(* Logix 5000 project; controller BreakGroup_US vendor 1 type 14 code 211 rev 32.16; software revision 32.05; part 5 of 8 *)
(* tags used below, declared in another part *)
   Emg_Stop : BOOL;
   Gantry_2_Tilter_LH_Start : BOOL;
   HMI_MAN_LH_OIL_STOP : BOOL;
   HMI_MAN_RH_OIL_STOP : BOOL;
   HMI_MAN_STN_100_STOP : BOOL;
   HMI_MAN_STN_110_STOP : BOOL;
   HMI_Oil_Tank_LH_PB : SINT;
   HMI_Oil_Tank_RH_PB : SINT;
   MAN_LH_OIL_TIME : TIMER;
   MAN_RH_OIL_TIME : TIMER;
   MAN_STN_100_HOME : TIMER;
   MAN_STN_110_HOME : TIMER;
   MCP_GY_01_Gripper : MCP_Servo_01;
   MCP_GY_01_Horizontal : MCP_Servo_02;
   MCP_GY_01_Vertical : MCP_Servo_02;
   RCP_LH_Oil_Tank_Lift : RCP_Servo_02;
   RCP_LH_Oil_Tank_Lift_Start : BOOL;
   RCP_RH_Oil_Tank_Lift : RCP_Servo_02;
   RCP_RH_Oil_Tank_Lift_Start : BOOL;
   RCP_ST_100_Turntable_Motor : RCP_Servo_02;
   RCP_ST_110_Turntable_Motor : RCP_Servo_02;
   ST10_Pre_Condition_OK : BOOL;
   ST10_Trolley1Lock_Cyl_01_Extended : ALIAS FOR MCP_PT01:1:I.0;
   ST10_Trolley1LockCyl_01_Retracted : ALIAS FOR MCP_PT01:1:I.1;
   ST10_Trolley_Present_Sensor : ALIAS FOR MCP_PT01:1:I.2;
   ST_100_Start : BOOL;
   ST_10_SEQ : DINT;
   ST_10_T1 : TIMER;
   ST_10_Trolley_FRWD : BOOL;
   ST_110_Start : BOOL;
   STN_100_Connection_Fault : BOOL;
   STN_100_Conveyor : INDEX_Block;
   STN_100_HMI_PB : SINT[2];
   STN_110_Connection_fault : BOOL;
   STN_110_Conveyor : INDEX_Block;
   STN_110_HMI_PB : SINT[2];

PROGRAM Oil_Tank_Lift   (* main routine Main *)

ROUTINE Main   (* ladder *)
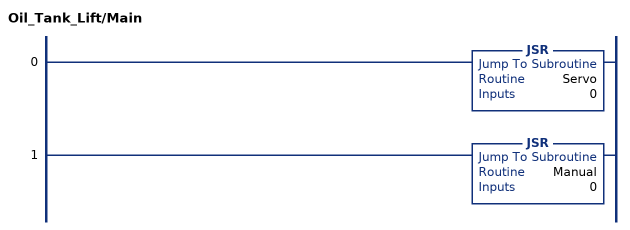
   0: JSR(Servo,0);
   1: JSR(Manual,0);
END_ROUTINE

ROUTINE Manual   (* ladder *)
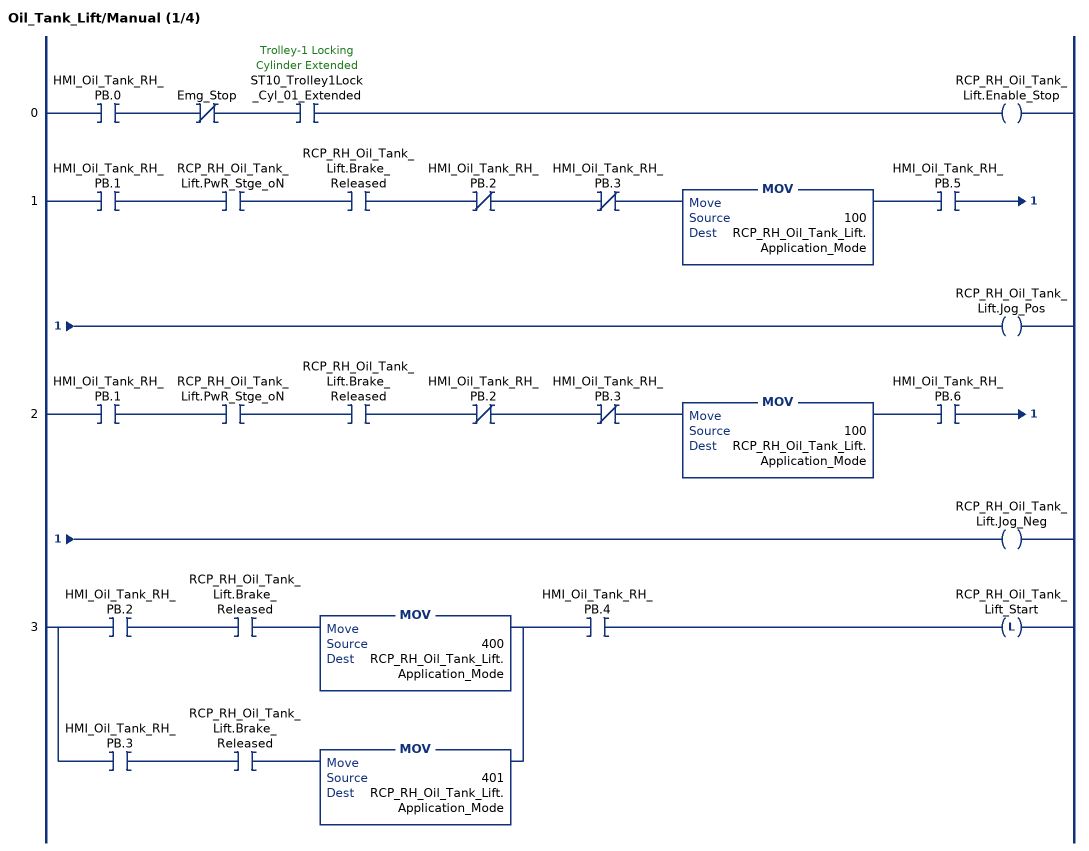
   0: XIC(HMI_Oil_Tank_RH_PB.0)XIO(Emg_Stop)XIC(ST10_Trolley1Lock_Cyl_01_Extended)OTE(RCP_RH_Oil_Tank_Lift.Enable_Stop);
   1: XIC(HMI_Oil_Tank_RH_PB.1)XIC(RCP_RH_Oil_Tank_Lift.PwR_Stge_oN)XIC(RCP_RH_Oil_Tank_Lift.Brake_Released)XIO(HMI_Oil_Tank_RH_PB.2)XIO(HMI_Oil_Tank_RH_PB.3)MOV(100,RCP_RH_Oil_Tank_Lift.Application_Mode)XIC(HMI_Oil_Tank_RH_PB.5)OTE(RCP_RH_Oil_Tank_Lift.Jog_Pos);
   2: XIC(HMI_Oil_Tank_RH_PB.1)XIC(RCP_RH_Oil_Tank_Lift.PwR_Stge_oN)XIC(RCP_RH_Oil_Tank_Lift.Brake_Released)XIO(HMI_Oil_Tank_RH_PB.2)XIO(HMI_Oil_Tank_RH_PB.3)MOV(100,RCP_RH_Oil_Tank_Lift.Application_Mode)XIC(HMI_Oil_Tank_RH_PB.6)OTE(RCP_RH_Oil_Tank_Lift.Jog_Neg);
   3: [XIC(HMI_Oil_Tank_RH_PB.2) XIC(RCP_RH_Oil_Tank_Lift.Brake_Released) MOV(400,RCP_RH_Oil_Tank_Lift.Application_Mode) ,XIC(HMI_Oil_Tank_RH_PB.3) XIC(RCP_RH_Oil_Tank_Lift.Brake_Released) MOV(401,RCP_RH_Oil_Tank_Lift.Application_Mode) ]XIC(HMI_Oil_Tank_RH_PB.4)OTL(RCP_RH_Oil_Tank_Lift_Start);
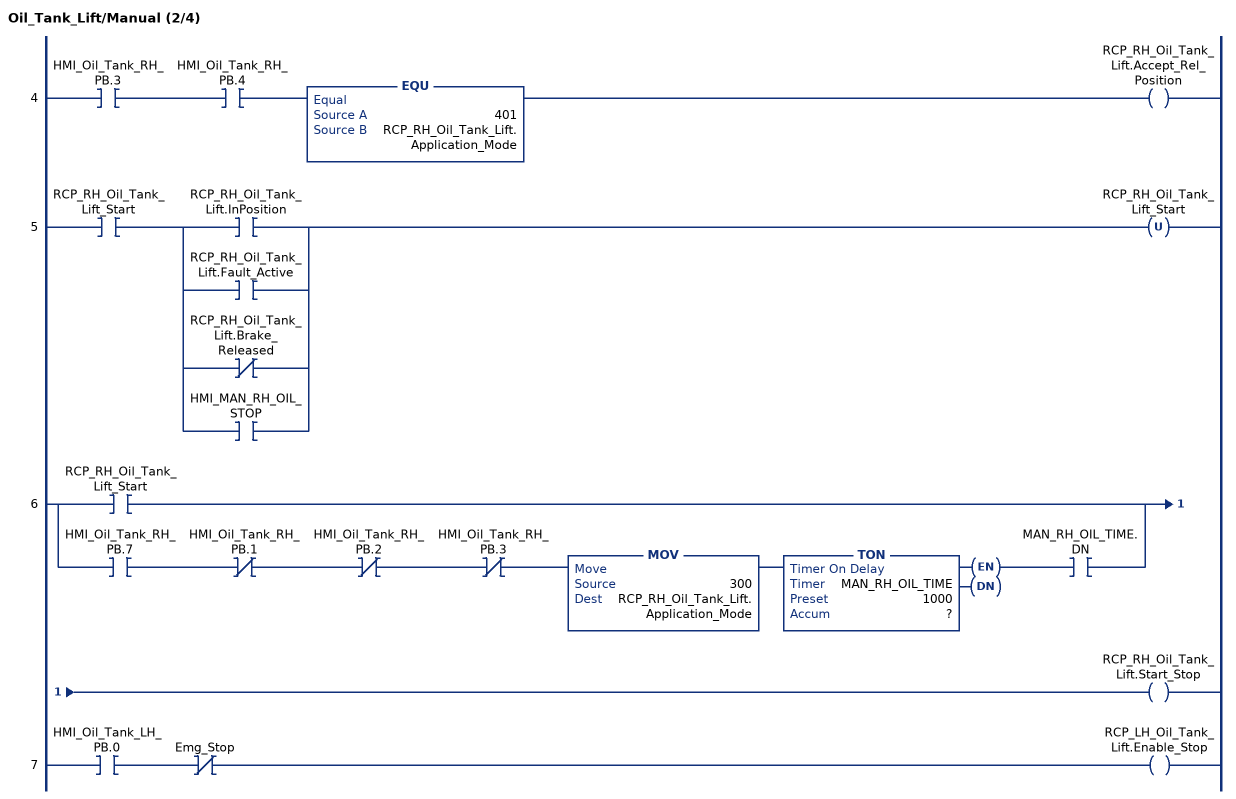
   4: XIC(HMI_Oil_Tank_RH_PB.3)XIC(HMI_Oil_Tank_RH_PB.4)EQU(401,RCP_RH_Oil_Tank_Lift.Application_Mode)OTE(RCP_RH_Oil_Tank_Lift.Accept_Rel_Position);
   5: XIC(RCP_RH_Oil_Tank_Lift_Start)[XIC(RCP_RH_Oil_Tank_Lift.InPosition) ,[XIC(RCP_RH_Oil_Tank_Lift.Fault_Active) ,[XIO(RCP_RH_Oil_Tank_Lift.Brake_Released) ,XIC(HMI_MAN_RH_OIL_STOP) ] ] ]OTU(RCP_RH_Oil_Tank_Lift_Start);
   6: [XIC(RCP_RH_Oil_Tank_Lift_Start) ,XIC(HMI_Oil_Tank_RH_PB.7) XIO(HMI_Oil_Tank_RH_PB.1) XIO(HMI_Oil_Tank_RH_PB.2) XIO(HMI_Oil_Tank_RH_PB.3) MOV(300,RCP_RH_Oil_Tank_Lift.Application_Mode) TON(MAN_RH_OIL_TIME,?,?) XIC(MAN_RH_OIL_TIME.DN) ]OTE(RCP_RH_Oil_Tank_Lift.Start_Stop);
   7: XIC(HMI_Oil_Tank_LH_PB.0)XIO(Emg_Stop)OTE(RCP_LH_Oil_Tank_Lift.Enable_Stop);
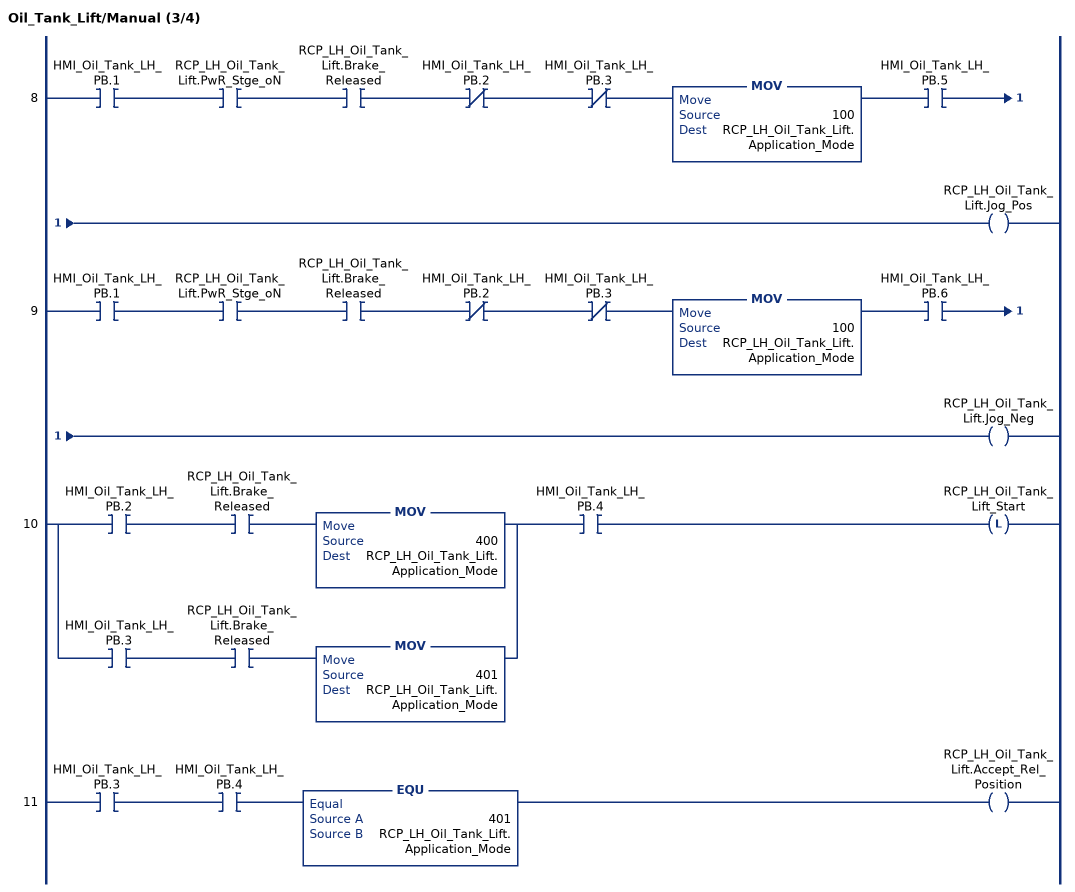
   8: XIC(HMI_Oil_Tank_LH_PB.1)XIC(RCP_LH_Oil_Tank_Lift.PwR_Stge_oN)XIC(RCP_LH_Oil_Tank_Lift.Brake_Released)XIO(HMI_Oil_Tank_LH_PB.2)XIO(HMI_Oil_Tank_LH_PB.3)MOV(100,RCP_LH_Oil_Tank_Lift.Application_Mode)XIC(HMI_Oil_Tank_LH_PB.5)OTE(RCP_LH_Oil_Tank_Lift.Jog_Pos);
   9: XIC(HMI_Oil_Tank_LH_PB.1)XIC(RCP_LH_Oil_Tank_Lift.PwR_Stge_oN)XIC(RCP_LH_Oil_Tank_Lift.Brake_Released)XIO(HMI_Oil_Tank_LH_PB.2)XIO(HMI_Oil_Tank_LH_PB.3)MOV(100,RCP_LH_Oil_Tank_Lift.Application_Mode)XIC(HMI_Oil_Tank_LH_PB.6)OTE(RCP_LH_Oil_Tank_Lift.Jog_Neg);
   10: [XIC(HMI_Oil_Tank_LH_PB.2) XIC(RCP_LH_Oil_Tank_Lift.Brake_Released) MOV(400,RCP_LH_Oil_Tank_Lift.Application_Mode) ,XIC(HMI_Oil_Tank_LH_PB.3) XIC(RCP_LH_Oil_Tank_Lift.Brake_Released) MOV(401,RCP_LH_Oil_Tank_Lift.Application_Mode) ]XIC(HMI_Oil_Tank_LH_PB.4)OTL(RCP_LH_Oil_Tank_Lift_Start);
   11: XIC(HMI_Oil_Tank_LH_PB.3)XIC(HMI_Oil_Tank_LH_PB.4)EQU(401,RCP_LH_Oil_Tank_Lift.Application_Mode)OTE(RCP_LH_Oil_Tank_Lift.Accept_Rel_Position);
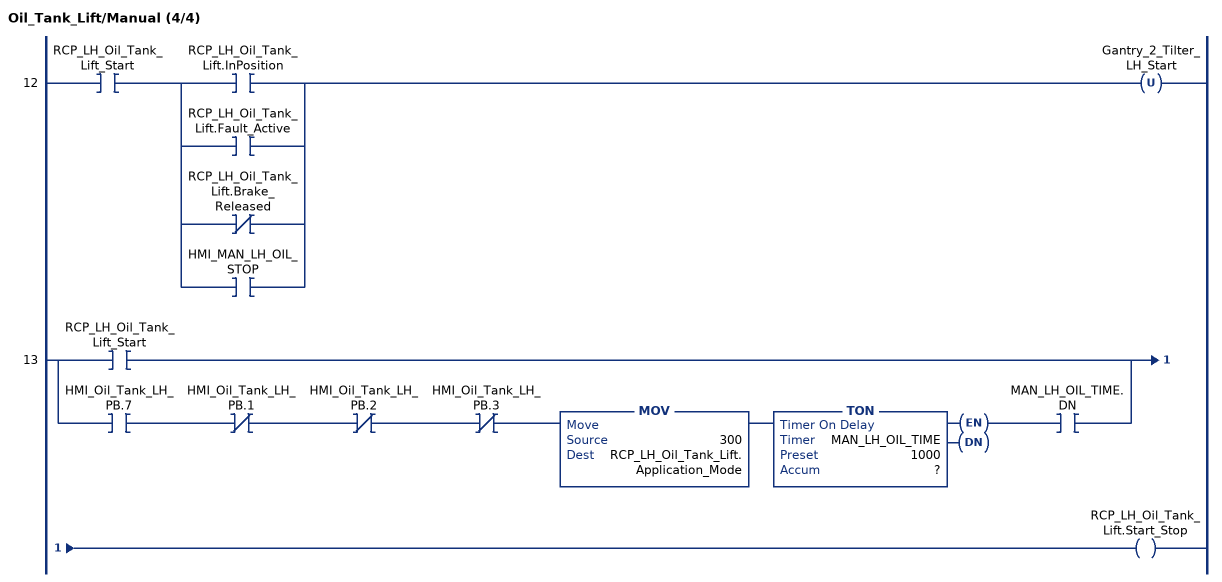
   12: XIC(RCP_LH_Oil_Tank_Lift_Start)[XIC(RCP_LH_Oil_Tank_Lift.InPosition) ,[XIC(RCP_LH_Oil_Tank_Lift.Fault_Active) ,[XIO(RCP_LH_Oil_Tank_Lift.Brake_Released) ,XIC(HMI_MAN_LH_OIL_STOP) ] ] ]OTU(Gantry_2_Tilter_LH_Start);
   13: [XIC(RCP_LH_Oil_Tank_Lift_Start) ,XIC(HMI_Oil_Tank_LH_PB.7) XIO(HMI_Oil_Tank_LH_PB.1) XIO(HMI_Oil_Tank_LH_PB.2) XIO(HMI_Oil_Tank_LH_PB.3) MOV(300,RCP_LH_Oil_Tank_Lift.Application_Mode) TON(MAN_LH_OIL_TIME,?,?) XIC(MAN_LH_OIL_TIME.DN) ]OTE(RCP_LH_Oil_Tank_Lift.Start_Stop);
END_ROUTINE

ROUTINE Servo   (* ladder *)
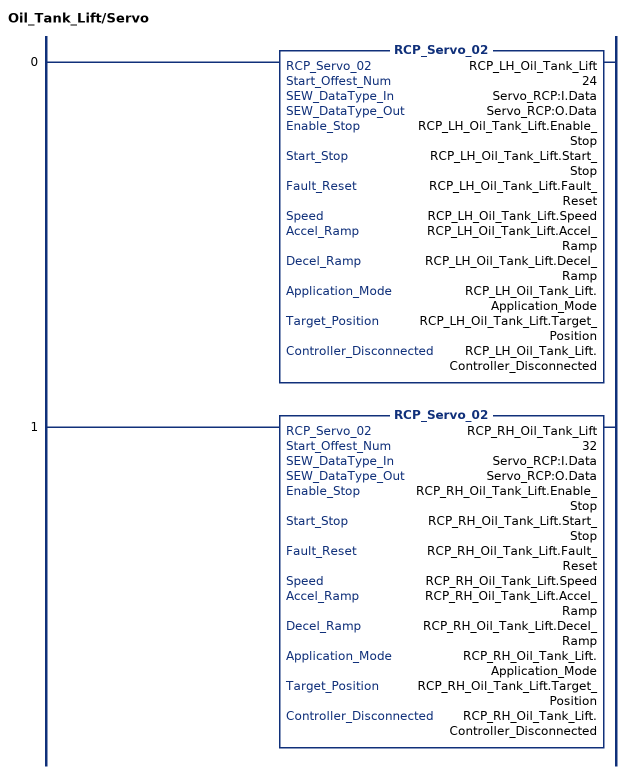
   0: RCP_Servo_02(RCP_LH_Oil_Tank_Lift,24,Servo_RCP:I.Data,Servo_RCP:O.Data,RCP_LH_Oil_Tank_Lift.Enable_Stop,RCP_LH_Oil_Tank_Lift.Start_Stop,RCP_LH_Oil_Tank_Lift.Fault_Reset,RCP_LH_Oil_Tank_Lift.Speed,RCP_LH_Oil_Tank_Lift.Accel_Ramp,RCP_LH_Oil_Tank_Lift.Decel_Ramp,RCP_LH_Oil_Tank_Lift.Application_Mode,RCP_LH_Oil_Tank_Lift.Target_Position,RCP_LH_Oil_Tank_Lift.Controller_Disconnected);
   1: RCP_Servo_02(RCP_RH_Oil_Tank_Lift,32,Servo_RCP:I.Data,Servo_RCP:O.Data,RCP_RH_Oil_Tank_Lift.Enable_Stop,RCP_RH_Oil_Tank_Lift.Start_Stop,RCP_RH_Oil_Tank_Lift.Fault_Reset,RCP_RH_Oil_Tank_Lift.Speed,RCP_RH_Oil_Tank_Lift.Accel_Ramp,RCP_RH_Oil_Tank_Lift.Decel_Ramp,RCP_RH_Oil_Tank_Lift.Application_Mode,RCP_RH_Oil_Tank_Lift.Target_Position,RCP_RH_Oil_Tank_Lift.Controller_Disconnected);
END_ROUTINE
END_PROGRAM

PROGRAM SafetyProgram   (* main routine MainRoutine, safety *)

ROUTINE MainRoutine   (* ladder *)
END_ROUTINE
END_PROGRAM

PROGRAM Station_10   (* main routine Main *)

ROUTINE Main   (* ladder *)
END_ROUTINE

ROUTINE Sequence   (* ladder *)
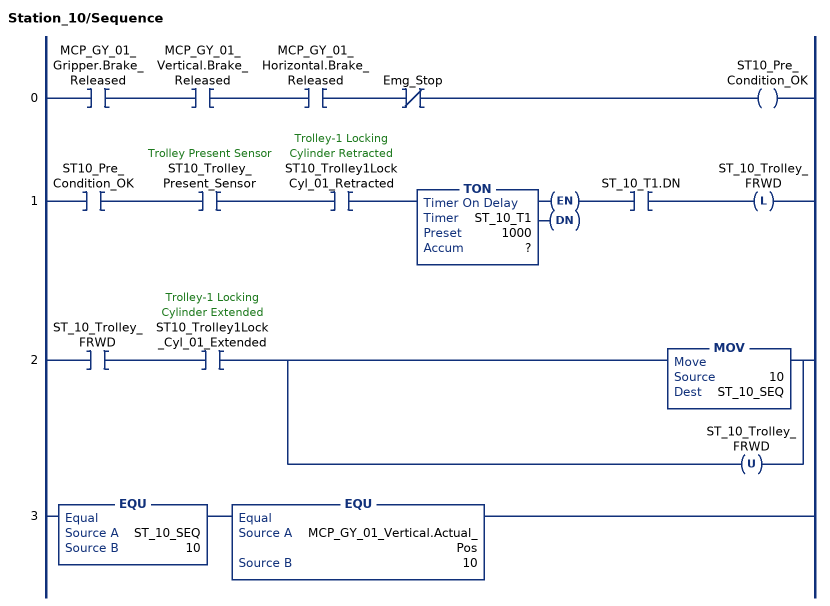
   0: XIC(MCP_GY_01_Gripper.Brake_Released)XIC(MCP_GY_01_Vertical.Brake_Released)XIC(MCP_GY_01_Horizontal.Brake_Released)XIO(Emg_Stop)OTE(ST10_Pre_Condition_OK);
   1: XIC(ST10_Pre_Condition_OK)XIC(ST10_Trolley_Present_Sensor)XIC(ST10_Trolley1LockCyl_01_Retracted)TON(ST_10_T1,?,?)XIC(ST_10_T1.DN)OTL(ST_10_Trolley_FRWD);
   2: XIC(ST_10_Trolley_FRWD)XIC(ST10_Trolley1Lock_Cyl_01_Extended)[MOV(10,ST_10_SEQ) ,OTU(ST_10_Trolley_FRWD) ];
   3: EQU(ST_10_SEQ,10)EQU(MCP_GY_01_Vertical.Actual_Pos,10);
END_ROUTINE
END_PROGRAM

PROGRAM Station_100   (* main routine Main *)

ROUTINE Main   (* ladder *)
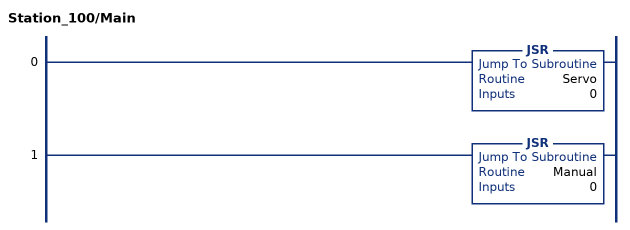
   0: JSR(Servo,0);
   1: JSR(Manual,0);
END_ROUTINE

ROUTINE Manual   (* ladder *)
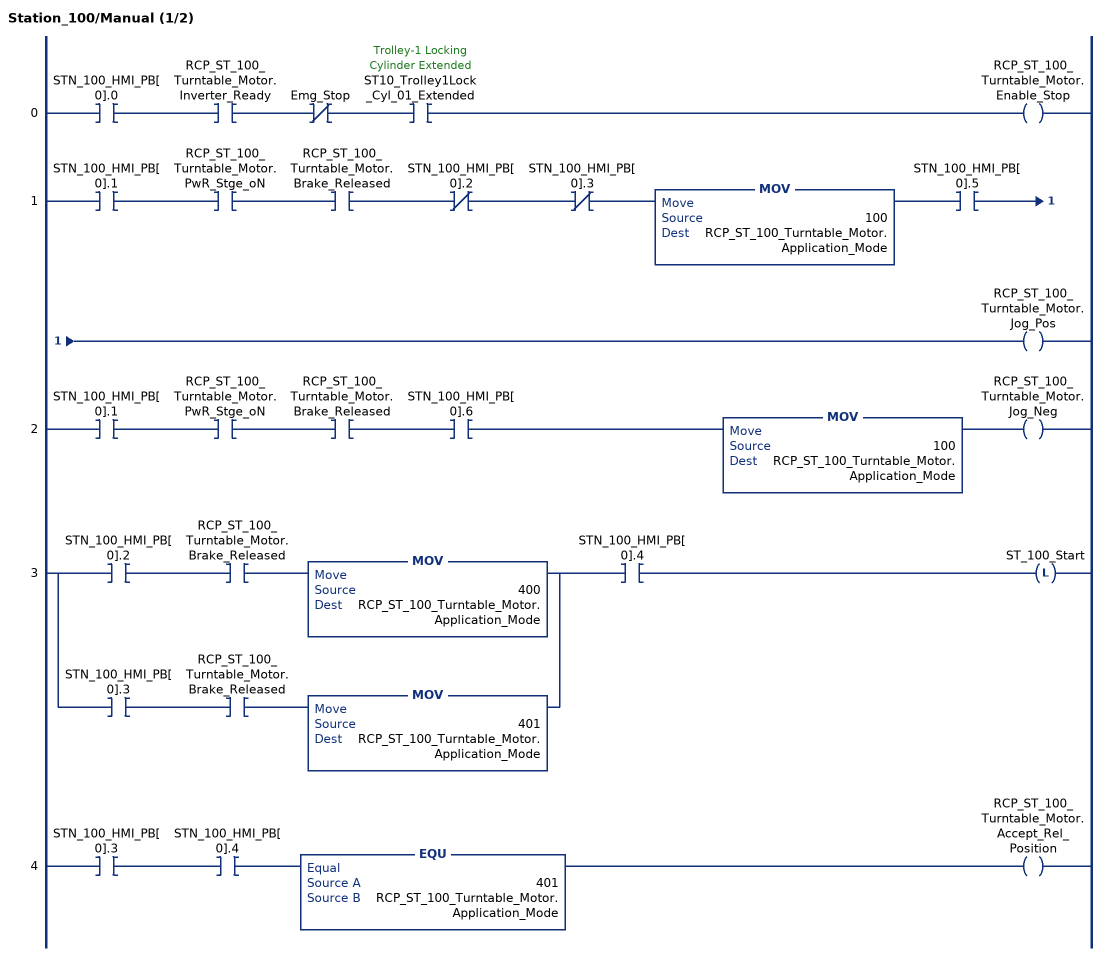
   0: XIC(STN_100_HMI_PB[0].0)XIC(RCP_ST_100_Turntable_Motor.Inverter_Ready)XIO(Emg_Stop)XIC(ST10_Trolley1Lock_Cyl_01_Extended)OTE(RCP_ST_100_Turntable_Motor.Enable_Stop);
   1: XIC(STN_100_HMI_PB[0].1)XIC(RCP_ST_100_Turntable_Motor.PwR_Stge_oN)XIC(RCP_ST_100_Turntable_Motor.Brake_Released)XIO(STN_100_HMI_PB[0].2)XIO(STN_100_HMI_PB[0].3)MOV(100,RCP_ST_100_Turntable_Motor.Application_Mode)XIC(STN_100_HMI_PB[0].5)OTE(RCP_ST_100_Turntable_Motor.Jog_Pos);
   2: XIC(STN_100_HMI_PB[0].1)XIC(RCP_ST_100_Turntable_Motor.PwR_Stge_oN)XIC(RCP_ST_100_Turntable_Motor.Brake_Released)XIC(STN_100_HMI_PB[0].6)MOV(100,RCP_ST_100_Turntable_Motor.Application_Mode)OTE(RCP_ST_100_Turntable_Motor.Jog_Neg);
   3: [XIC(STN_100_HMI_PB[0].2) XIC(RCP_ST_100_Turntable_Motor.Brake_Released) MOV(400,RCP_ST_100_Turntable_Motor.Application_Mode) ,XIC(STN_100_HMI_PB[0].3) XIC(RCP_ST_100_Turntable_Motor.Brake_Released) MOV(401,RCP_ST_100_Turntable_Motor.Application_Mode) ]XIC(STN_100_HMI_PB[0].4)OTL(ST_100_Start);
   4: XIC(STN_100_HMI_PB[0].3)XIC(STN_100_HMI_PB[0].4)EQU(401,RCP_ST_100_Turntable_Motor.Application_Mode)OTE(RCP_ST_100_Turntable_Motor.Accept_Rel_Position);
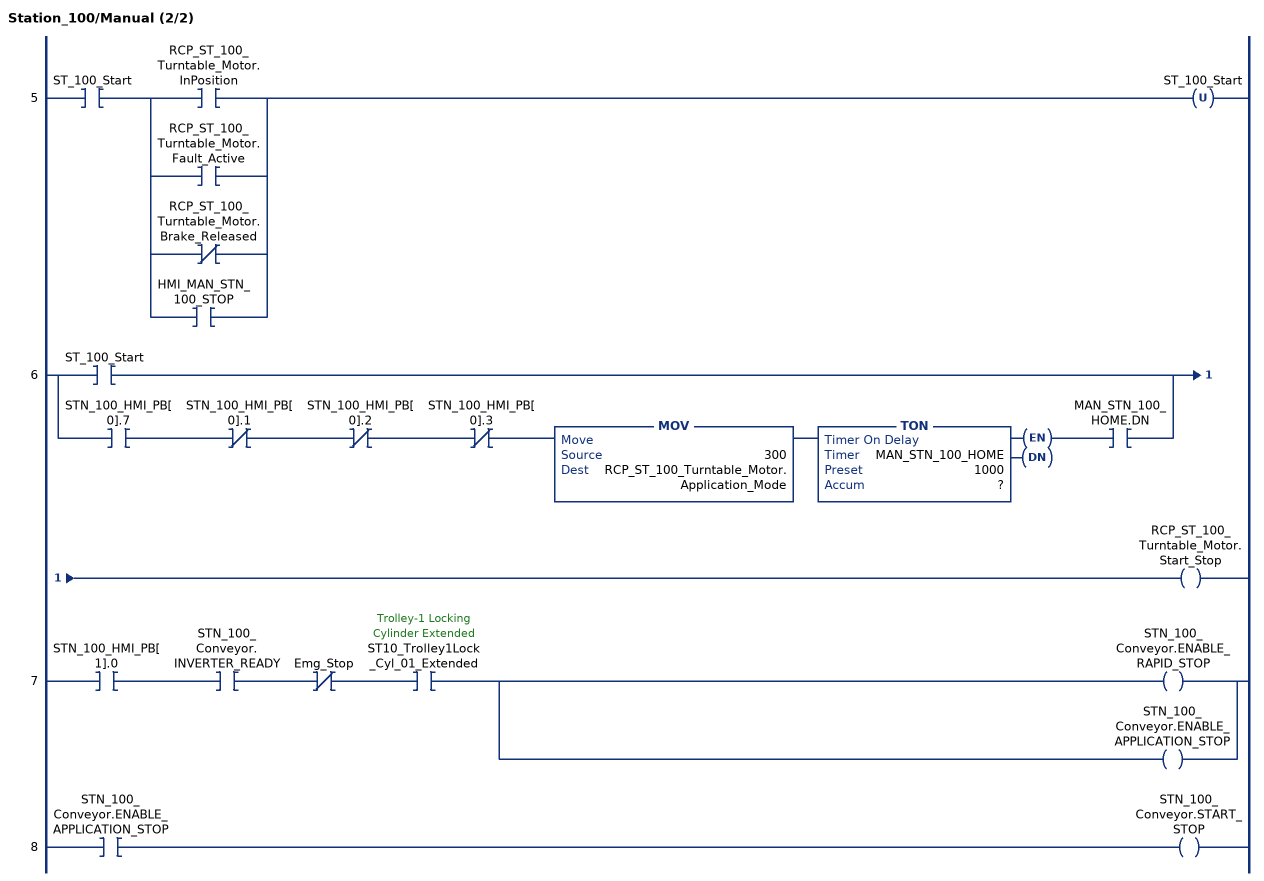
   5: XIC(ST_100_Start)[XIC(RCP_ST_100_Turntable_Motor.InPosition) ,[XIC(RCP_ST_100_Turntable_Motor.Fault_Active) ,[XIO(RCP_ST_100_Turntable_Motor.Brake_Released) ,XIC(HMI_MAN_STN_100_STOP) ] ] ]OTU(ST_100_Start);
   6: [XIC(ST_100_Start) ,XIC(STN_100_HMI_PB[0].7) XIO(STN_100_HMI_PB[0].1) XIO(STN_100_HMI_PB[0].2) XIO(STN_100_HMI_PB[0].3) MOV(300,RCP_ST_100_Turntable_Motor.Application_Mode) TON(MAN_STN_100_HOME,?,?) XIC(MAN_STN_100_HOME.DN) ]OTE(RCP_ST_100_Turntable_Motor.Start_Stop);
   7: XIC(STN_100_HMI_PB[1].0)XIC(STN_100_Conveyor.INVERTER_READY)XIO(Emg_Stop)XIC(ST10_Trolley1Lock_Cyl_01_Extended)[OTE(STN_100_Conveyor.ENABLE_RAPID_STOP) ,OTE(STN_100_Conveyor.ENABLE_APPLICATION_STOP) ];
   8: XIC(STN_100_Conveyor.ENABLE_APPLICATION_STOP)OTE(STN_100_Conveyor.START_STOP);
END_ROUTINE

ROUTINE Servo   (* ladder *)
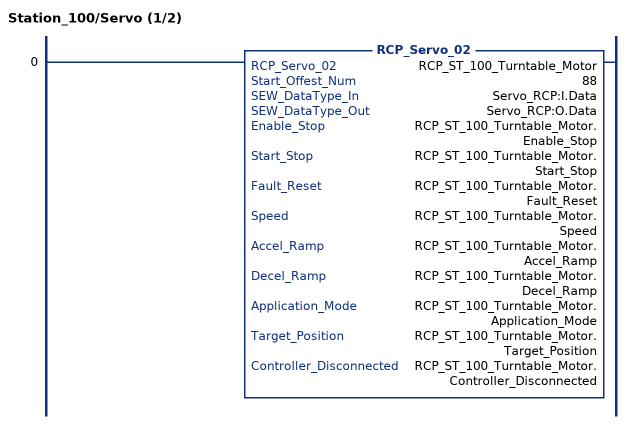
   0: RCP_Servo_02(RCP_ST_100_Turntable_Motor,88,Servo_RCP:I.Data,Servo_RCP:O.Data,RCP_ST_100_Turntable_Motor.Enable_Stop,RCP_ST_100_Turntable_Motor.Start_Stop,RCP_ST_100_Turntable_Motor.Fault_Reset,RCP_ST_100_Turntable_Motor.Speed,RCP_ST_100_Turntable_Motor.Accel_Ramp,RCP_ST_100_Turntable_Motor.Decel_Ramp,RCP_ST_100_Turntable_Motor.Application_Mode,RCP_ST_100_Turntable_Motor.Target_Position,RCP_ST_100_Turntable_Motor.Controller_Disconnected);
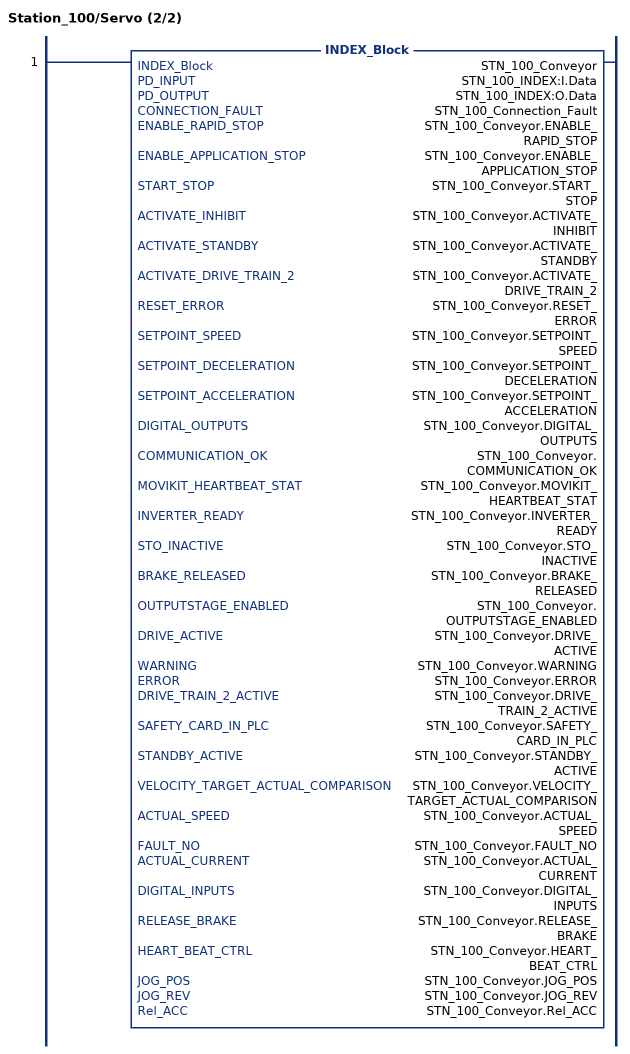
   1: INDEX_Block(STN_100_Conveyor,STN_100_INDEX:I.Data,STN_100_INDEX:O.Data,STN_100_Connection_Fault,STN_100_Conveyor.ENABLE_RAPID_STOP,STN_100_Conveyor.ENABLE_APPLICATION_STOP,STN_100_Conveyor.START_STOP,STN_100_Conveyor.ACTIVATE_INHIBIT,STN_100_Conveyor.ACTIVATE_STANDBY,STN_100_Conveyor.ACTIVATE_DRIVE_TRAIN_2,STN_100_Conveyor.RESET_ERROR,STN_100_Conveyor.SETPOINT_SPEED,STN_100_Conveyor.SETPOINT_DECELERATION,STN_100_Conveyor.SETPOINT_ACCELERATION,STN_100_Conveyor.DIGITAL_OUTPUTS,STN_100_Conveyor.COMMUNICATION_OK,STN_100_Conveyor.MOVIKIT_HEARTBEAT_STAT,STN_100_Conveyor.INVERTER_READY,STN_100_Conveyor.STO_INACTIVE,STN_100_Conveyor.BRAKE_RELEASED,STN_100_Conveyor.OUTPUTSTAGE_ENABLED,STN_100_Conveyor.DRIVE_ACTIVE,STN_100_Conveyor.WARNING,STN_100_Conveyor.ERROR,STN_100_Conveyor.DRIVE_TRAIN_2_ACTIVE,STN_100_Conveyor.SAFETY_CARD_IN_PLC,STN_100_Conveyor.STANDBY_ACTIVE,STN_100_Conveyor.VELOCITY_TARGET_ACTUAL_COMPARISON,STN_100_Conveyor.ACTUAL_SPEED,STN_100_Conveyor.FAULT_NO,STN_100_Conveyor.ACTUAL_CURRENT,STN_100_Conveyor.DIGITAL_INPUTS,STN_100_Conveyor.RELEASE_BRAKE,STN_100_Conveyor.HEART_BEAT_CTRL,STN_100_Conveyor.JOG_POS,STN_100_Conveyor.JOG_REV,STN_100_Conveyor.Rel_ACC);
END_ROUTINE
END_PROGRAM

PROGRAM Station_110   (* main routine Main *)

ROUTINE Main   (* ladder *)
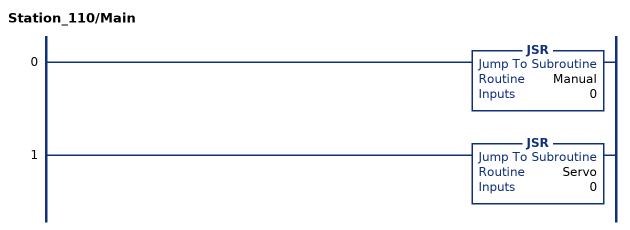
   0: JSR(Manual,0);
   1: JSR(Servo,0);
END_ROUTINE

ROUTINE Manual   (* ladder *)
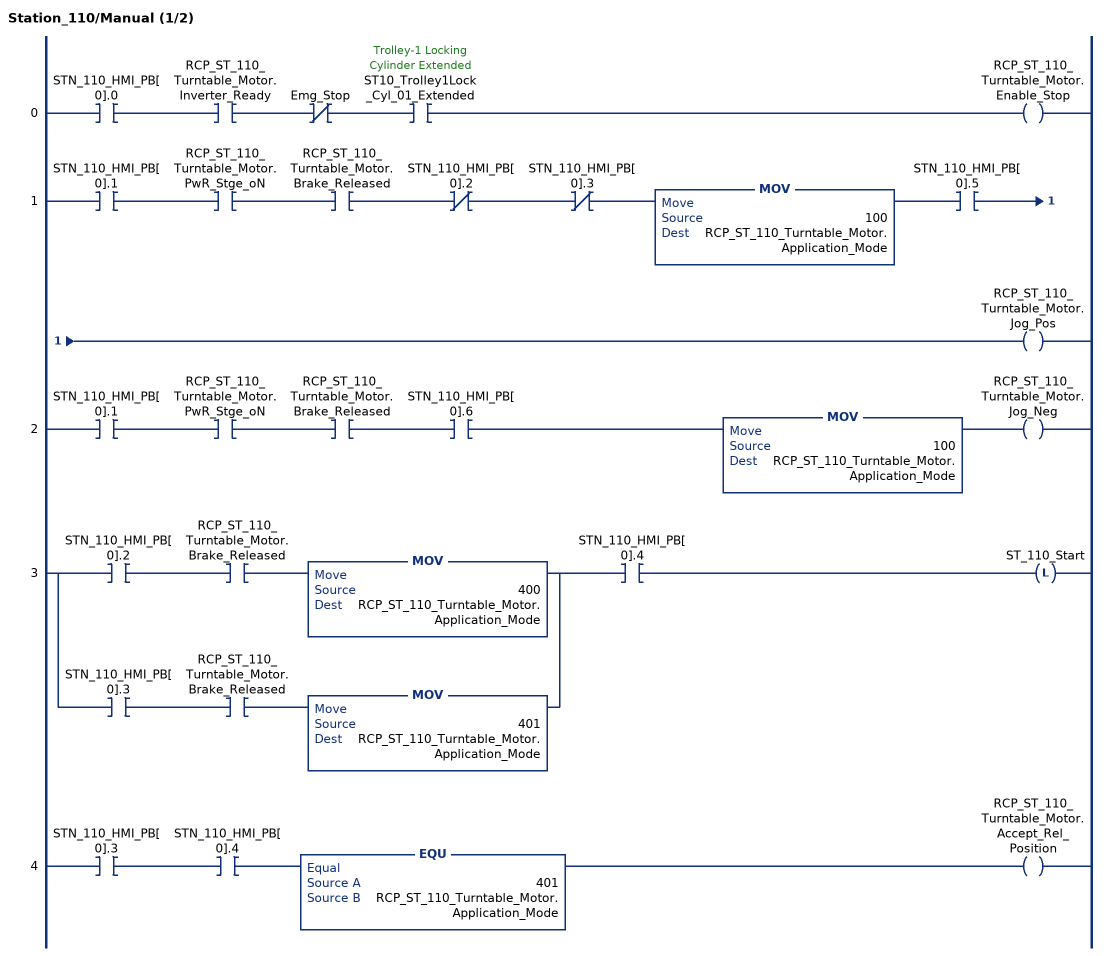
   0: XIC(STN_110_HMI_PB[0].0)XIC(RCP_ST_110_Turntable_Motor.Inverter_Ready)XIO(Emg_Stop)XIC(ST10_Trolley1Lock_Cyl_01_Extended)OTE(RCP_ST_110_Turntable_Motor.Enable_Stop);
   1: XIC(STN_110_HMI_PB[0].1)XIC(RCP_ST_110_Turntable_Motor.PwR_Stge_oN)XIC(RCP_ST_110_Turntable_Motor.Brake_Released)XIO(STN_110_HMI_PB[0].2)XIO(STN_110_HMI_PB[0].3)MOV(100,RCP_ST_110_Turntable_Motor.Application_Mode)XIC(STN_110_HMI_PB[0].5)OTE(RCP_ST_110_Turntable_Motor.Jog_Pos);
   2: XIC(STN_110_HMI_PB[0].1)XIC(RCP_ST_110_Turntable_Motor.PwR_Stge_oN)XIC(RCP_ST_110_Turntable_Motor.Brake_Released)XIC(STN_110_HMI_PB[0].6)MOV(100,RCP_ST_110_Turntable_Motor.Application_Mode)OTE(RCP_ST_110_Turntable_Motor.Jog_Neg);
   3: [XIC(STN_110_HMI_PB[0].2) XIC(RCP_ST_110_Turntable_Motor.Brake_Released) MOV(400,RCP_ST_110_Turntable_Motor.Application_Mode) ,XIC(STN_110_HMI_PB[0].3) XIC(RCP_ST_110_Turntable_Motor.Brake_Released) MOV(401,RCP_ST_110_Turntable_Motor.Application_Mode) ]XIC(STN_110_HMI_PB[0].4)OTL(ST_110_Start);
   4: XIC(STN_110_HMI_PB[0].3)XIC(STN_110_HMI_PB[0].4)EQU(401,RCP_ST_110_Turntable_Motor.Application_Mode)OTE(RCP_ST_110_Turntable_Motor.Accept_Rel_Position);
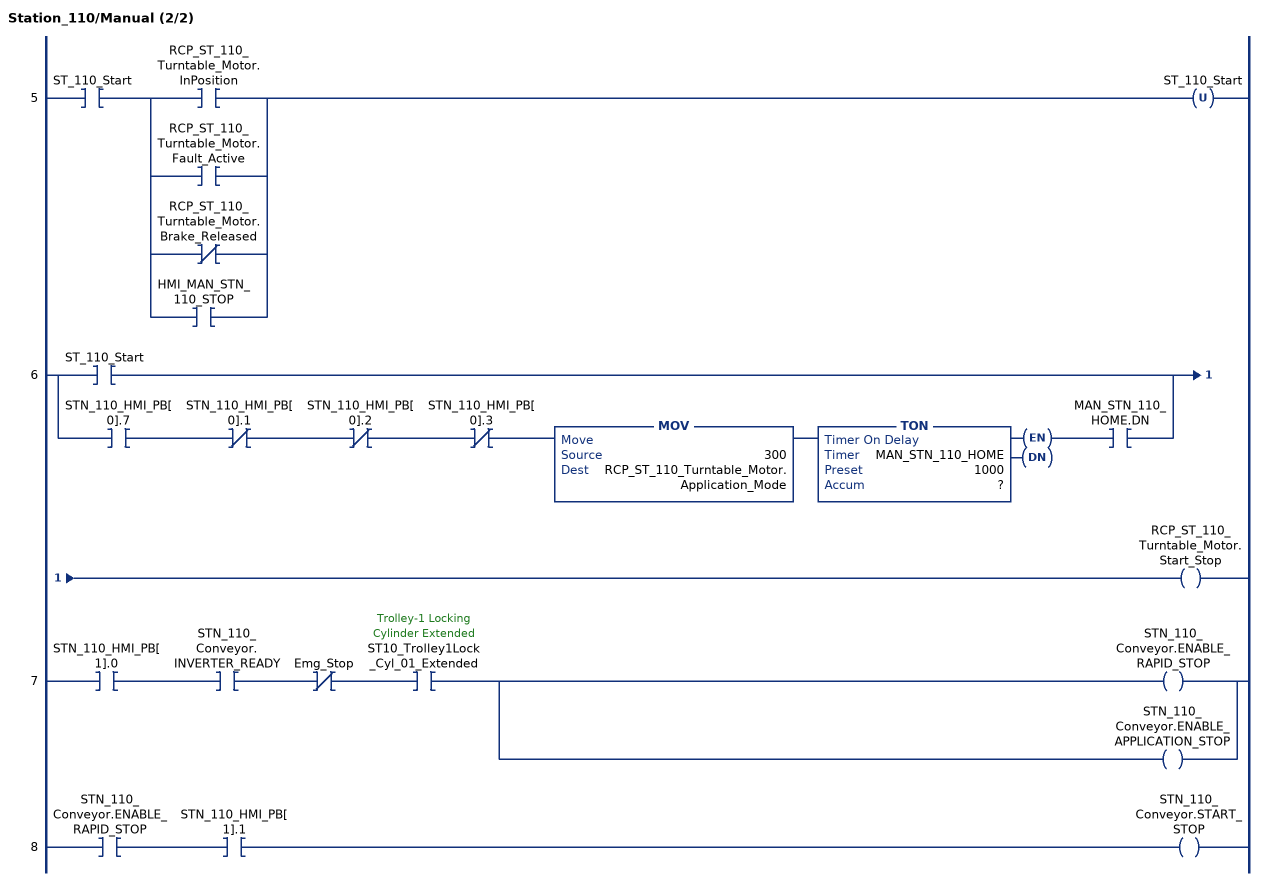
   5: XIC(ST_110_Start)[XIC(RCP_ST_110_Turntable_Motor.InPosition) ,[XIC(RCP_ST_110_Turntable_Motor.Fault_Active) ,[XIO(RCP_ST_110_Turntable_Motor.Brake_Released) ,XIC(HMI_MAN_STN_110_STOP) ] ] ]OTU(ST_110_Start);
   6: [XIC(ST_110_Start) ,XIC(STN_110_HMI_PB[0].7) XIO(STN_110_HMI_PB[0].1) XIO(STN_110_HMI_PB[0].2) XIO(STN_110_HMI_PB[0].3) MOV(300,RCP_ST_110_Turntable_Motor.Application_Mode) TON(MAN_STN_110_HOME,?,?) XIC(MAN_STN_110_HOME.DN) ]OTE(RCP_ST_110_Turntable_Motor.Start_Stop);
   7: XIC(STN_110_HMI_PB[1].0)XIC(STN_110_Conveyor.INVERTER_READY)XIO(Emg_Stop)XIC(ST10_Trolley1Lock_Cyl_01_Extended)[OTE(STN_110_Conveyor.ENABLE_RAPID_STOP) ,OTE(STN_110_Conveyor.ENABLE_APPLICATION_STOP) ];
   8: XIC(STN_110_Conveyor.ENABLE_RAPID_STOP)XIC(STN_110_HMI_PB[1].1)OTE(STN_110_Conveyor.START_STOP);
END_ROUTINE

ROUTINE Servo   (* ladder *)
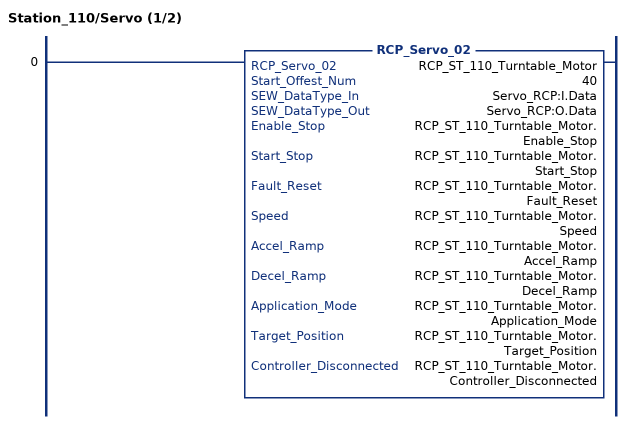
   0: RCP_Servo_02(RCP_ST_110_Turntable_Motor,40,Servo_RCP:I.Data,Servo_RCP:O.Data,RCP_ST_110_Turntable_Motor.Enable_Stop,RCP_ST_110_Turntable_Motor.Start_Stop,RCP_ST_110_Turntable_Motor.Fault_Reset,RCP_ST_110_Turntable_Motor.Speed,RCP_ST_110_Turntable_Motor.Accel_Ramp,RCP_ST_110_Turntable_Motor.Decel_Ramp,RCP_ST_110_Turntable_Motor.Application_Mode,RCP_ST_110_Turntable_Motor.Target_Position,RCP_ST_110_Turntable_Motor.Controller_Disconnected);
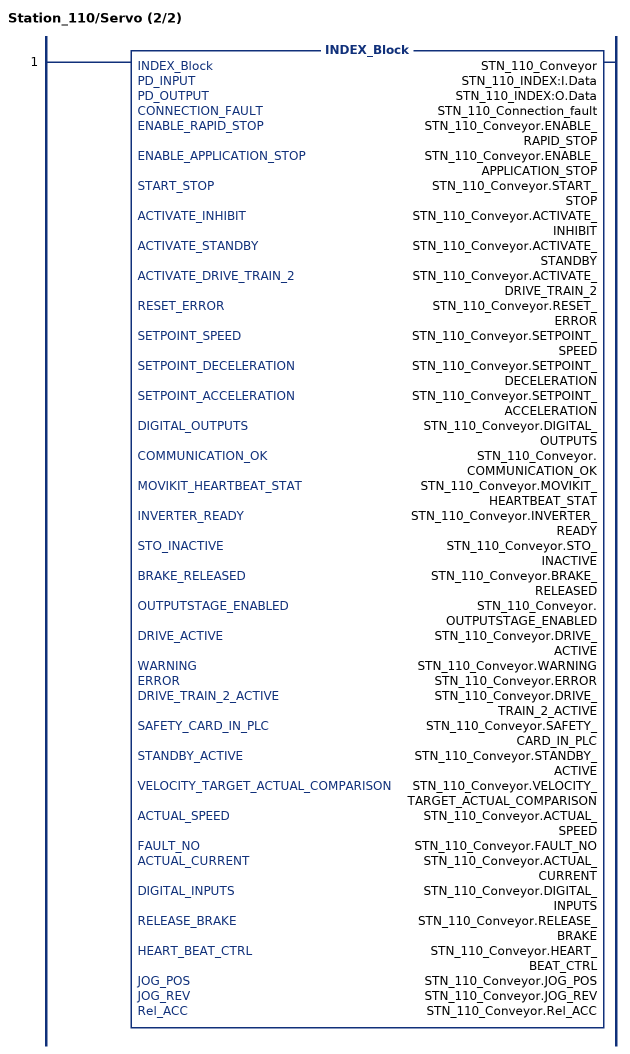
   1: INDEX_Block(STN_110_Conveyor,STN_110_INDEX:I.Data,STN_110_INDEX:O.Data,STN_110_Connection_fault,STN_110_Conveyor.ENABLE_RAPID_STOP,STN_110_Conveyor.ENABLE_APPLICATION_STOP,STN_110_Conveyor.START_STOP,STN_110_Conveyor.ACTIVATE_INHIBIT,STN_110_Conveyor.ACTIVATE_STANDBY,STN_110_Conveyor.ACTIVATE_DRIVE_TRAIN_2,STN_110_Conveyor.RESET_ERROR,STN_110_Conveyor.SETPOINT_SPEED,STN_110_Conveyor.SETPOINT_DECELERATION,STN_110_Conveyor.SETPOINT_ACCELERATION,STN_110_Conveyor.DIGITAL_OUTPUTS,STN_110_Conveyor.COMMUNICATION_OK,STN_110_Conveyor.MOVIKIT_HEARTBEAT_STAT,STN_110_Conveyor.INVERTER_READY,STN_110_Conveyor.STO_INACTIVE,STN_110_Conveyor.BRAKE_RELEASED,STN_110_Conveyor.OUTPUTSTAGE_ENABLED,STN_110_Conveyor.DRIVE_ACTIVE,STN_110_Conveyor.WARNING,STN_110_Conveyor.ERROR,STN_110_Conveyor.DRIVE_TRAIN_2_ACTIVE,STN_110_Conveyor.SAFETY_CARD_IN_PLC,STN_110_Conveyor.STANDBY_ACTIVE,STN_110_Conveyor.VELOCITY_TARGET_ACTUAL_COMPARISON,STN_110_Conveyor.ACTUAL_SPEED,STN_110_Conveyor.FAULT_NO,STN_110_Conveyor.ACTUAL_CURRENT,STN_110_Conveyor.DIGITAL_INPUTS,STN_110_Conveyor.RELEASE_BRAKE,STN_110_Conveyor.HEART_BEAT_CTRL,STN_110_Conveyor.JOG_POS,STN_110_Conveyor.JOG_REV,STN_110_Conveyor.Rel_ACC);
END_ROUTINE
END_PROGRAM

PROGRAM Station_120   (* main routine Main *)

ROUTINE Main   (* ladder *)
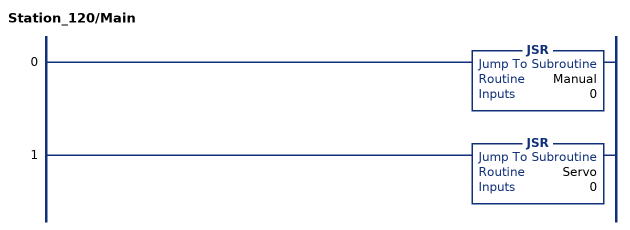
   0: JSR(Manual,0);
   1: JSR(Servo,0);
END_ROUTINE
